FUNCTION_BLOCK FB_CommandChangeUnSuspend EXTENDS FB_CommandChange IMPLEMENTS ITF_CommandChange
VAR

END_VAR

METHOD Execute : BOOL
VAR_INPUT
END_VAR
END_METHOD

END_FUNCTION_BLOCK

(* stored: Version 1.1.0.1
   POU FB_CommandChangeUnSuspend: Id {03c9589a-fc15-0c4a-14e8-fb8dbfc85e4c}, SpecialFunc None
   Method Execute: Id {af28a0de-e214-001a-3556-df82a40ec4e4} *)
